FUNCTION_BLOCK FB_RC_Servo_Test EXTENDS TcUnit.FB_TestSuite

// SetpointReached();
// Stop();

METHOD PRIVATE OutputRamped
VAR_INPUT
END_VAR
END_METHOD

METHOD PRIVATE SetpointChanged
VAR_INPUT
END_VAR
END_METHOD

METHOD SetpointReached
VAR
	Servo : FB_RC_Servo;
	Setpoint : INT := 10;
	ExpectedSetpointReached : INT := 10;
	Result : INT;
END_VAR
TEST('TEST: Setpoint reached');

Servo(stop := FALSE,
	setpoint := Setpoint,
	rampSpeed := 10,
	trapezoidalProfileActive := FALSE,
	servoAngleMin := 0,
	servoAngleMax := 100,
	rampCycleTime := T#1MS,
	currentPositionSetpoint => Result);
	


AssertEquals(Expected := ExpectedSetpointReached,
	Actual := Servo.currentPositionSetpoint,
	Message := 'Expected value not reached');

TEST_FINISHED();
END_METHOD

METHOD PRIVATE StartingPosition
VAR_INPUT
END_VAR
END_METHOD

METHOD PRIVATE Stop
VAR
	stop : BOOL;
	init1 : BOOL := TRUE;
	init2 : BOOL := TRUE;
	init3 : BOOL := TRUE;
	intermediateVal1 : INT;
	intermediateVal2 : INT;
	valuesAreEqualAndNotZero : BOOL := FALSE;
	startValue : INT := 0;
	setpoint : INT := 10000;
	minValue : INT := 0;
	maxValue : INT := 10000;
	cycleTime : TIME := T#1MS;
	rampSpeed : INT := 20;
	FB_Servo: FB_RC_Servo;
	timer1: TON;
	timer2: TON;
	ExpectedValue : BOOL := TRUE;
END_VAR
IF init1 THEN
	stop := FALSE;
	init1 := FALSE;
END_IF;

timer1(IN:= TRUE, PT:= T#1000S, Q=> , ET=> );
timer2(IN:= TRUE, PT:= T#1000S, Q=> , ET=> );

FB_Servo(
	stop:= stop, 
	setpoint:= setpoint, 
	rampSpeed:= rampSpeed, 
	trapezoidalProfileActive:= FALSE, 
	servoAngleMin:= minValue, 
	servoAngleMax:= maxValue, 
	rampCycleTime:= cycleTime, 
	rampStartPos:= startValue, 
	currentPositionSetpoint=> , 
	error=> );

IF timer1.ET > T#1S AND init2 THEN
	stop := TRUE;
	intermediateVal1 := FB_Servo.currentPositionSetpoint;
	init2 := FALSE;
END_IF

IF timer2.ET > T#2S AND init3 THEN
	IF intermediateVal1 = intermediateVal2 AND intermediateVal1 <> 0 THEN
		valuesAreEqualAndNotZero := TRUE;
	END_IF
END_IF

AssertEquals(
Expected:= ExpectedValue,
 Actual:= valuesAreEqualAndNotZero,
 Message:= 'Ramp was not stopped or value was not ramped');
END_METHOD

METHOD PRIVATE Trapezoidal
VAR_INPUT
END_VAR
END_METHOD

END_FUNCTION_BLOCK

(* stored: Version 1.1.0.1, ProductVersion 3.1.4024.13
   POU FB_RC_Servo_Test: Id {03ef9bed-a740-4d16-836d-7c880d928d4f}, SpecialFunc None
   Method OutputRamped: Id {557fe578-98bf-49e6-93fd-344654483c78}
   Method SetpointChanged: Id {36afbb44-edb3-4ebd-b626-09555da2a097}
   Method SetpointReached: Id {8b035494-74d9-4637-aeda-8bb4b708ea31}
   Method StartingPosition: Id {bae9910b-fa54-4115-b0d1-420fbae8a281}
   Method Stop: Id {85fc3fb1-42c1-4b4e-80db-93ea81d1e0b1}
   Method Trapezoidal: Id {f76f3628-c236-4862-a00d-cdcbd1386b7e} *)
